TYPE DUT_SENSOR_DATAS_3 :
UNION
	data_lreal:REAL;
	data_byte:ARRAY[0..3] OF BYTE;
END_UNION
END_TYPE

(* stored: Version 1.1.0.1, ProductVersion 3.1.4024.6
   DUT DUT_SENSOR_DATAS_3: Id {c16abbbb-e4c2-4992-8318-fbb99781d0f8} *)
